{attribute 'pack_mode' := '1'}
    {attribute 'OPC.UA.DA' := '1'}
    {attribute 'OPC.UA.DA.StructuredType' := '1'}
    (*
    ST_RWToPLC_HMI_IgnitionExp
    ==================================================
    Generated from Ignition UDT: RW_ToPLC
    Total tags: 2
    Generated on: 2025-09-15 12:47:19
    *)
    TYPE ST_RWToPLC_HMI_IgnitionExp :
    STRUCT
        {attribute 'OPC.UA.DA' := '1'}
        {attribute 'OPC.UA.DA.Description' := '{Description}'}
        // {Description}
        Value : REAL := 0.0;
        {attribute 'OPC.UA.DA' := '1'}
        {attribute 'OPC.UA.DA.Access' := '1'}
        Reference : REAL := 0.0;		// Read-only tag
    END_STRUCT
    END_TYPE

(* stored: Version 1.1.0.1
   DUT ST_RWToPLC_HMI_IgnitionExp: Id {8149f486-260b-4749-ab1b-e2a074eeb093} *)
